FUNCTION_BLOCK EL2252
VAR
	{attribute addProperty Name "WcState"}
	_wcState : WcStateBase;
	{attribute addProperty Name "Info data"}
	_infoData : InfoDataDC;
	_io : EL2252_Data;
END_VAR

PROPERTY IO : REFERENCE TO EL2252_Data
GET
IO REF= _io;
END_GET
END_PROPERTY

PROPERTY WcState : REFERENCE TO WcStateBase
GET
WcState REF= _wcState;
END_GET
END_PROPERTY

END_FUNCTION_BLOCK

(* stored: Version 1.1.0.1, ProductVersion 3.1.4024.9
   POU EL2252: Id {b70986d3-5337-04f9-1022-1f990c4ef203}, SpecialFunc None
   Property IO: Id {aedd889d-3515-0a9e-09b0-1c889e479b85}
   Get Get: Id {471d8ac7-09a5-0134-0f57-1ee419b9cdea}
   Property WcState: Id {7b7b30f2-95bc-0da6-3b70-4b36c0022196}
   Get Get: Id {8eaf57ad-d1c0-0c92-227d-cb22cdfd7e60} *)
